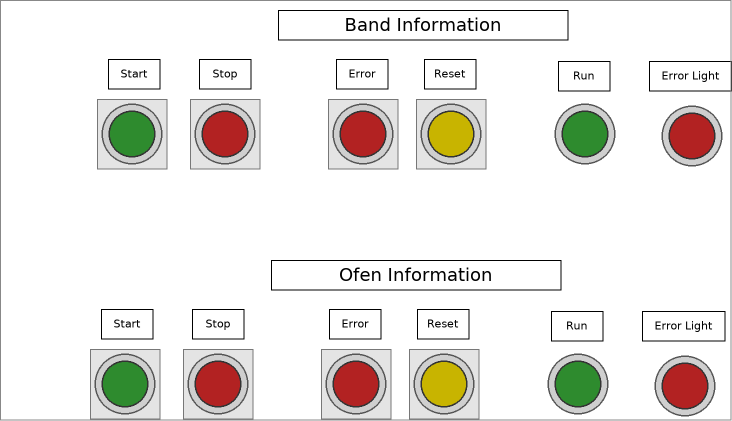
VISUALIZATION Visualization  // 732x421
    PushSwitch (97,99 70x70), variable: MAIN.bBandStart, behaviour: TOGGLE, style: Switch-PushSwitch-Green
    PushSwitch (190,99 70x70), variable: MAIN.bBandStop, behaviour: TOGGLE, style: Switch-PushSwitch-Red
    PushSwitch (328,99 70x70), variable: MAIN.bBandErr, behaviour: TOGGLE, style: Switch-PushSwitch-Red
    PushSwitch (416,99 70x70), variable: MAIN.bBandReset, behaviour: TOGGLE, style: Switch-PushSwitch-Yellow
    Lamp1 (550,99 70x70), variable: MAIN.fbBandMotor.bMotorRun, style: Lamp-Lamp1-Green
    Lamp1 (657,101 70x70), variable: MAIN.fbBandMotor.bErrorLight, style: Lamp-Lamp1-Red
    Rectangle (108,59 52x30), "Start"
    Rectangle (199,59 52x30), "Stop"
    Rectangle (336,59 52x30), "Error"
    Rectangle (424,59 52x30), "Reset"
    Rectangle (558,61 52x30), "Run"
    Rectangle (649,61 83x30), "Error Light"
    Rectangle (278,10 290x30), "Band Information"
    PushSwitch (90,349 70x70), variable: MAIN.bOfenStart, behaviour: TOGGLE, style: Switch-PushSwitch-Green
    PushSwitch (183,349 70x70), variable: MAIN.bOfenStop, behaviour: TOGGLE, style: Switch-PushSwitch-Red
    PushSwitch (321,349 70x70), variable: MAIN.bOfenErr, behaviour: TOGGLE, style: Switch-PushSwitch-Red
    PushSwitch (409,349 70x70), variable: MAIN.bOfenReset, behaviour: TOGGLE, style: Switch-PushSwitch-Yellow
    Lamp1 (543,349 70x70), variable: MAIN.fbOfenMotor.bMotorRun, style: Lamp-Lamp1-Green
    Lamp1 (650,351 70x70), variable: MAIN.fbOfenMotor.bErrorLight, style: Lamp-Lamp1-Red
    Rectangle (101,309 52x30), "Start"
    Rectangle (192,309 52x30), "Stop"
    Rectangle (329,309 52x30), "Error"
    Rectangle (417,309 52x30), "Reset"
    Rectangle (551,311 52x30), "Run"
    Rectangle (642,311 83x30), "Error Light"
    Rectangle (271,260 290x30), "Ofen Information"
END_VISUALIZATION

(* stored: Version 1.1.0.1
   Visu Visualization: Id {364b7a09-312f-46c2-b7be-5de5ff742dab} *)
